SUBAPPLICATION Inputs (* Subapplication Type *)
  (* Standard: 61499-2 *)
  (* Version 1.0, 2025-01-31, franz *)
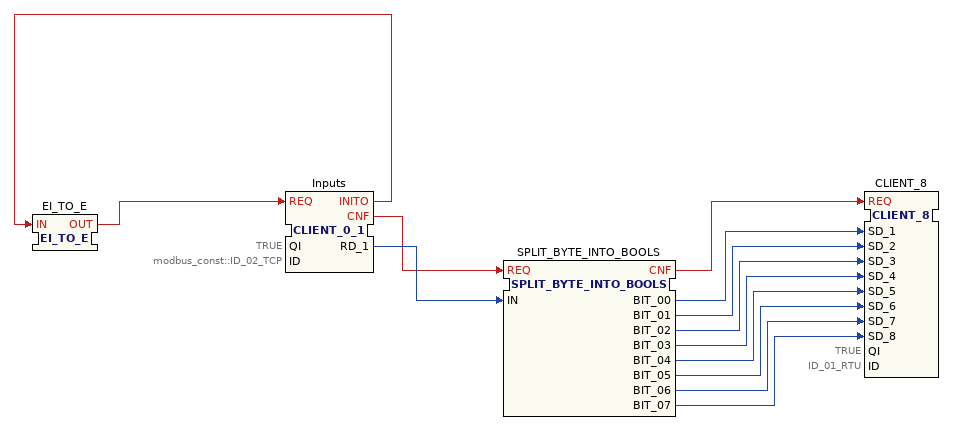
  FBS
    SPLIT_BYTE_INTO_BOOLS : SPLIT_BYTE_INTO_BOOLS;
    Inputs : CLIENT_0_1(QI := TRUE, ID := modbus_const::ID_02_TCP);
    EI_TO_E : EI_TO_E;
    CLIENT_8 : CLIENT_8(QI := TRUE, ID := ID_01_RTU);
  END_FBS
  EVENT_CONNECTIONS
    Inputs.INITO TO EI_TO_E.IN;
    EI_TO_E.OUT TO Inputs.REQ;
    Inputs.CNF TO SPLIT_BYTE_INTO_BOOLS.REQ;
    SPLIT_BYTE_INTO_BOOLS.CNF TO CLIENT_8.REQ;
  END_CONNECTIONS
  DATA_CONNECTIONS
    Inputs.RD_1 TO SPLIT_BYTE_INTO_BOOLS.IN;
    SPLIT_BYTE_INTO_BOOLS.BIT_00 TO CLIENT_8.SD_1;
    SPLIT_BYTE_INTO_BOOLS.BIT_01 TO CLIENT_8.SD_2;
    SPLIT_BYTE_INTO_BOOLS.BIT_02 TO CLIENT_8.SD_3;
    SPLIT_BYTE_INTO_BOOLS.BIT_03 TO CLIENT_8.SD_4;
    SPLIT_BYTE_INTO_BOOLS.BIT_04 TO CLIENT_8.SD_5;
    SPLIT_BYTE_INTO_BOOLS.BIT_05 TO CLIENT_8.SD_6;
    SPLIT_BYTE_INTO_BOOLS.BIT_06 TO CLIENT_8.SD_7;
    SPLIT_BYTE_INTO_BOOLS.BIT_07 TO CLIENT_8.SD_8;
  END_CONNECTIONS
END_SUBAPPLICATION
